{attribute addProperty BoxType "EJ7342-0000-0019"}
{attribute addProperty Id "ENC_Status_compact_ChannelAT %I*ARRAY[0..1] OF ENC_Status_compact_Channel_559DED9896120DCM_Status_ChannelAT %I*ARRAY[0..1] OF DCM_Status_Channel_C2B0CAE13240ENC_Control_compact_ChannelAT %Q*ARRAY[0..1] OF ENC_Control_compact_Channel_5C86AA9D6480DCM_Control_Channel_1AT %Q*DCM_Control_Channel_6F24B2C41620DCM_Velocity_Channel_1AT %Q*DCM_Velocity_Channel_1D89B5C21620DCM_Control_Channel_2AT %Q*DCM_Control_Channel_6F24B2C41620DCM_Velocity_Channel_2AT %Q*DCM_Velocity_Channel_1D89B5C21620WcStateAT %I*WcState_F855686C1620InfoDataAT %I*InfoData_3F3BB279112140"}
{attribute addProperty CRC "2530475426"}
{attribute addProperty SizeInBites "384"}
{attribute addProperty SizeInBytes "48"}
TYPE EJ7342_5DC6D752 :
STRUCT
	{attribute addProperty Name "ENC_Status_compact_Channel"}
	ENC_Status_compact_Channel : ARRAY[0..1] OF ENC_Status_compact_Channel_559DED98;
	{attribute addProperty Name "DCM_Status_Channel"}
	DCM_Status_Channel : ARRAY[0..1] OF DCM_Status_Channel_C2B0CAE1;
	{attribute addProperty Name "ENC_Control_compact_Channel"}
	ENC_Control_compact_Channel : ARRAY[0..1] OF ENC_Control_compact_Channel_5C86AA9D;
	{attribute addProperty Name "DCM_Control_Channel_1"}
	DCM_Control_Channel_1 : DCM_Control_Channel_6F24B2C4;
	{attribute addProperty Name "DCM_Velocity_Channel_1"}
	DCM_Velocity_Channel_1 : DCM_Velocity_Channel_1D89B5C2;
	{attribute addProperty Name "DCM_Control_Channel_2"}
	DCM_Control_Channel_2 : DCM_Control_Channel_6F24B2C4;
	{attribute addProperty Name "DCM_Velocity_Channel_2"}
	DCM_Velocity_Channel_2 : DCM_Velocity_Channel_1D89B5C2;
	{attribute addProperty Name "WcState"}
	WcState : WcState_F855686C;
	{attribute addProperty Name "InfoData"}
	InfoData : InfoData_3F3BB279;
END_STRUCT
END_TYPE

(* stored: Version 1.2.0.0, ProductVersion 3.1.4024.9
   DUT EJ7342_5DC6D752: Id {a8037808-0991-4bf3-bd92-82f1881b9cdd} *)
